Staubli VAL3: onEdit.pgx

public program onEdit(string& x_sItem[])
  local num l_nResult
  local num i
  local string l_sItem
  local string l_sType
begin
  //
  // go to the view instruction page
  //
  if size(x_sItem)==1
    // show the items
    if isDefined(saveProg:pProg[x_sItem].iEvent)
      for i=0 to size(saveProg:pProg[x_sItem].iEvent)-1
        l_sItem=l_sItem+saveProg:pProg[x_sItem].iEvent[i].sType+" "+saveProg:pProg[x_sItem].iEvent[i].sData +chr(10)
      endFor
      // remove the last CR
      l_sItem=left(l_sItem,len(l_sItem)-1)
      // show IT
      popUpMsg(l_sItem)
    endIf
  else
    call getType(l_sType)
    saveData:sProgTypeUsing=l_sType
    // load it
    call load(x_sItem,l_nResult)
    // give it back
    x_sItem[1]=x_sItem
    x_sItem="Disk://instruction/PROG/page_instr"
  endIf
end
